TYPE Mat35 : ARRAY[1..3, 1..5] OF LREAL; END_TYPE

(* stored: Version 1.1.0.1, ProductVersion 3.1.4024.11
   DUT Mat35: Id {e3d0fc9e-bbd3-40a9-87e3-55689651abcc} *)
